{attribute addProperty BoxType "ER7342-0002-0021"}
{attribute addProperty Id "ENC_Status_compact_ChannelAT %I*ARRAY[0..1] OF ENC_Status_compact_Channel_A7E8355C96120DCM_Status_ChannelAT %I*ARRAY[0..1] OF DCM_Status_Channel_64D937433240ENC_Control_compact_ChannelAT %Q*ARRAY[0..1] OF ENC_Control_compact_Channel_5C86AA9D6480DCM_Control_Channel_1AT %Q*DCM_Control_Channel_6F24B2C41620DCM_Velocity_Channel_1AT %Q*DCM_Velocity_Channel_1D89B5C21620DCM_Control_Channel_2AT %Q*DCM_Control_Channel_6F24B2C41620DCM_Velocity_Channel_2AT %Q*DCM_Velocity_Channel_1D89B5C21620WcStateAT %I*WcState_98A4DF7520.250InfoDataAT %I*InfoData_3F3BB279112140"}
{attribute addProperty CRC "873791271"}
{attribute addProperty SizeInBites "370"}
{attribute addProperty SizeInBytes "46.25"}
TYPE ER7342_E2585B83 :
STRUCT
	{attribute addProperty Name "ENC_Status_compact_Channel"}
	ENC_Status_compact_Channel : ARRAY[0..1] OF ENC_Status_compact_Channel_A7E8355C;
	{attribute addProperty Name "DCM_Status_Channel"}
	DCM_Status_Channel : ARRAY[0..1] OF DCM_Status_Channel_64D93743;
	{attribute addProperty Name "ENC_Control_compact_Channel"}
	ENC_Control_compact_Channel : ARRAY[0..1] OF ENC_Control_compact_Channel_5C86AA9D;
	{attribute addProperty Name "DCM_Control_Channel_1"}
	DCM_Control_Channel_1 : DCM_Control_Channel_6F24B2C4;
	{attribute addProperty Name "DCM_Velocity_Channel_1"}
	DCM_Velocity_Channel_1 : DCM_Velocity_Channel_1D89B5C2;
	{attribute addProperty Name "DCM_Control_Channel_2"}
	DCM_Control_Channel_2 : DCM_Control_Channel_6F24B2C4;
	{attribute addProperty Name "DCM_Velocity_Channel_2"}
	DCM_Velocity_Channel_2 : DCM_Velocity_Channel_1D89B5C2;
	{attribute addProperty Name "WcState"}
	WcState : WcState_98A4DF75;
	{attribute addProperty Name "InfoData"}
	InfoData : InfoData_3F3BB279;
END_STRUCT
END_TYPE

(* stored: Version 1.2.0.0, ProductVersion 3.1.4024.9
   DUT ER7342_E2585B83: Id {d9a612c7-1caa-4ef5-aea8-7ce6d25fbb79} *)
